(* PLC project Unnamed, Unknown Unnamed 1 *)
(* stored: creationDateTime 2012-09-12T23:30:19, modificationDateTime 2015-06-18T11:28:47 *)

PROGRAM main
  VAR_EXTERNAL
    Power_ON : BOOL;
    Power_OFF : BOOL;
    power : BOOL;
    DrawTest : BOOL;
    DrawLogo : BOOL;
    DrawEscher : BOOL;
    Detect_Circle : BOOL;
  END_VAR
  VAR
    RS0 : RS;
  END_VAR

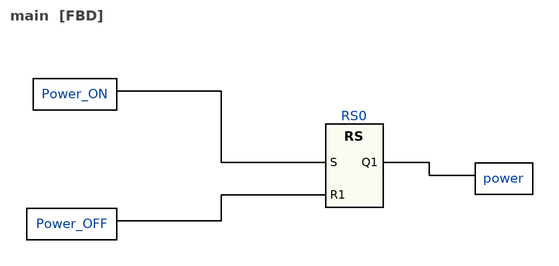
(* FBD diagram, written out as Structured Text *)
RS0(S := Power_ON, R1 := Power_OFF);
power := RS0.Q1;
END_PROGRAM

PROGRAM ReadGUIdata
  VAR
    tmp : INT;
  END_VAR
  VAR_EXTERNAL
    power : BOOL;
    XaxisPos : INT;
    YaxisPos : INT;
    ZaxisPos : INT;
    TaxisPos : INT;
  END_VAR

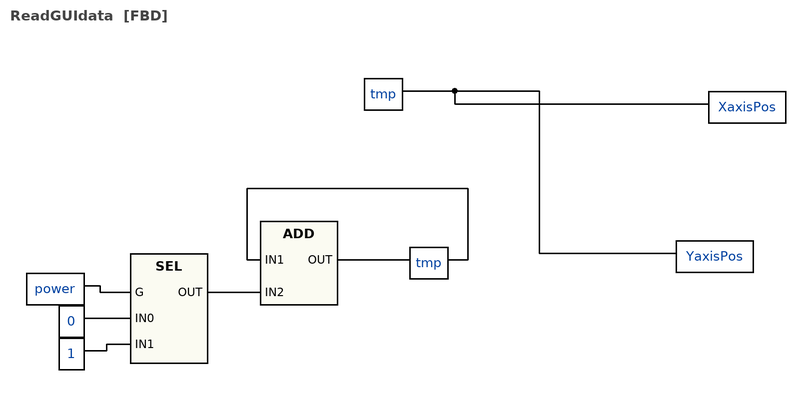
(* FBD diagram, written out as Structured Text *)
XaxisPos := tmp;
tmp := tmp + SEL(power, 0, 1);
YaxisPos := tmp;
END_PROGRAM

PROGRAM Declarations
  VAR
    LocalVar0 : DINT;
    LocalVar1 : DINT;
  END_VAR

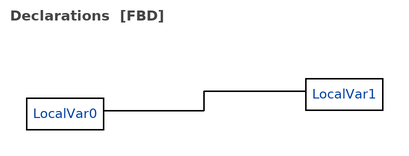
(* FBD diagram, written out as Structured Text *)
LocalVar1 := LocalVar0;
END_PROGRAM

CONFIGURATION config
  RESOURCE resource1 ON PLC
    VAR_GLOBAL
      Initialize : BOOL := TRUE;
      power : BOOL := TRUE;
    END_VAR
    TASK InitOneShot(SINGLE := Initialize, PRIORITY := 0);
    TASK ControlTask(INTERVAL := T#2ms, PRIORITY := 0);
    TASK GUIupdate(INTERVAL := T#40ms, PRIORITY := 0);
    PROGRAM Initializer WITH InitOneShot : Declarations;
    PROGRAM MainInstance WITH ControlTask : main;
    PROGRAM PosReader WITH GUIupdate : ReadGUIdata;
  END_RESOURCE
END_CONFIGURATION
